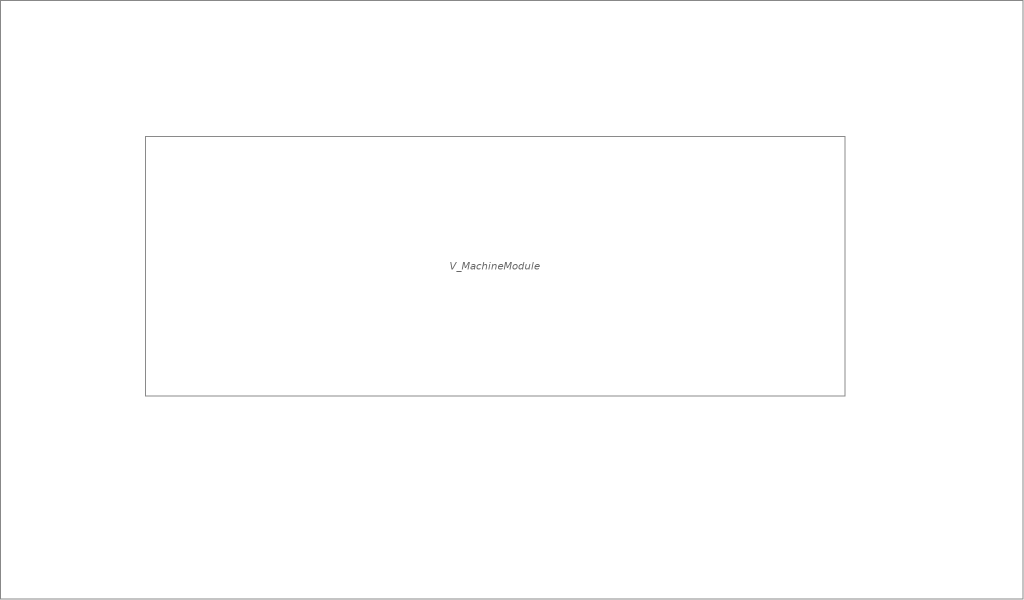
VISUALIZATION V_Main  // 1024x600
    Frame (145,136 700x260)
        shows V_MachineModule(HMI := MAIN.Seedra.PackMLBaseModule_HMI)
END_VISUALIZATION

(* stored: Version 1.1.0.1
   Visu V_Main: Id {a820fc1e-d71f-479f-a200-f2cc0d18dc0b} *)
